// TIA Portal V15 export
// export: Created 2018-12-31T00:40:19.1865532Z, ExportSetting WithDefaults, WithReadOnly, DisplayName Totally Integrated Automation Portal, DisplayVersion V15 Update 2, DisplayName TIA Portal Openness, DisplayVersion V15 Update 2, DisplayName STEP 7 Professional, DisplayVersion V15 Update 2, DisplayName STEP 7 Safety, DisplayVersion V15, DisplayName WinCC Professional, DisplayVersion V15 Update 2, DisplayName SIMATIC Visualization Architect, DisplayVersion V15 Update 1
TYPE "iUDT_PI_ADRxx34_APPL_ROBNAME"
// stored: CreationDate 2017-02-22T17:41:39.0757837Z, InterfaceModifiedDate 2017-05-29T07:23:13.1164474Z, IsConsistent true, IsKnowHowProtected false, LibraryConformanceStatus The object is library-conformant., ModifiedDate 2018-01-29T16:41:32.9213311Z
   STRUCT
      "RB-PLC" : Struct   // RB-PLC interlocks
      END_STRUCT;
      "RB-RB" : Struct   // RB-RB interlock signal
      END_STRUCT;
   END_STRUCT;
END_TYPE
